Universal Robots PolyScope program: 10_return_home.urp

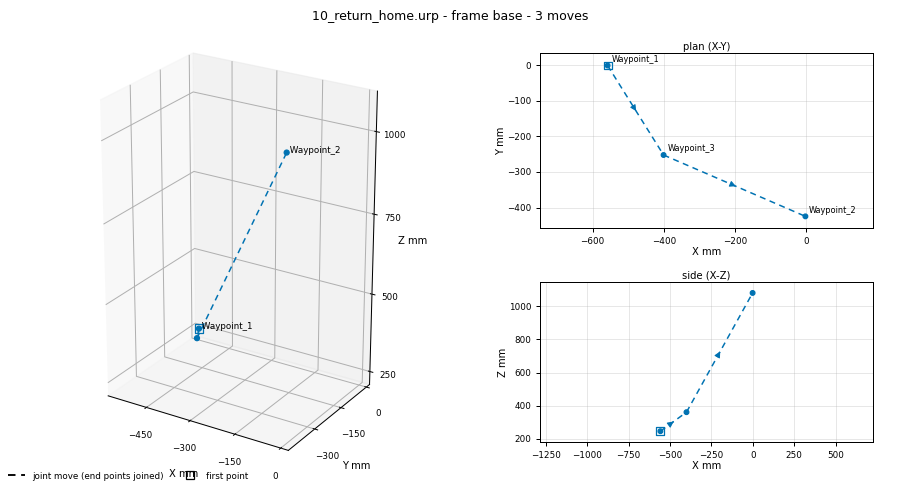
[picture p0: tool path of 10_return_home.urp in frame base, 3 of 3 moves have a stored position in this frame; points joined in program order, loops and branches not executed]
Program 10_return_home (installation=default directory=/programs/washer_rahman createdIn=5.9.5.1031259 lastSavedIn=5.9.5.1031259 robotSerialNumber=20215500597)
Calibrated DH parameters: a=[0.000193, -0.066673, -0.391568, -0.000012, 0.00005, 0]; d=[0.162643, -472.05677, 465.132521, 7.058239, 0.099746, 0.099582]; alpha=[1.571116, 0.00089, 0.003862, 1.569269, -1.569248, 0]; deltaTheta=[0, -1.413394, 7.628392, 0.068187, 0, -0.000001]
Robot Program (runOnlyOnce=true)
  SuppressedNode
    Script: glass_hover=p[-.603,-0.23+GP_int_in[0]*0.150 ,0.277,2.067,2.652,-2.043]
  MoveJ speed 60 deg/s, acceleration 80 deg/s^2 (useActiveTCP=true) feature=Base
    Waypoint Waypoint_1: TCP in base x=-557.946 y=-0.629 z=246.472 mm, rx=-1.2337 ry=-1.2229 rz=1.2356 rad; joints [-31.234, -63.253, 147.704, -263.237, -57.851, 1.051] deg; TCP offset x=0 y=0 z=191.5 mm, rx=0 ry=0 rz=0 rad
    Waypoint Waypoint_3: TCP in base x=-400.494 y=-252.295 z=361.215 mm, rx=-0.4201 ry=-1.9938 rz=1.9794 rad; joints [-31.194, -86.068, 141.579, -237.45, 6.863, 1.527] deg
    SuppressedNode
      Waypoint hover1: TCP in base x=-557.942 y=-0.628 z=246.464 mm, rx=-1.2338 ry=-1.2229 rz=1.2356 rad; joints [-31.234, -63.251, 147.705, -263.24, -57.851, 1.053] deg
    MoveJ speed 60 deg/s, acceleration 80 deg/s^2 (useActiveTCP=true) feature=Base
      Waypoint Waypoint_2: TCP in base x=-1.607 y=-424.817 z=1080.554 mm, rx=-0.0045 ry=-2.2185 rz=2.2204 rad; joints [-0.001, -89.997, 0, -89.999, -0.001, -0.002] deg
